RoboDK station: UR5Trajectory1.rdk

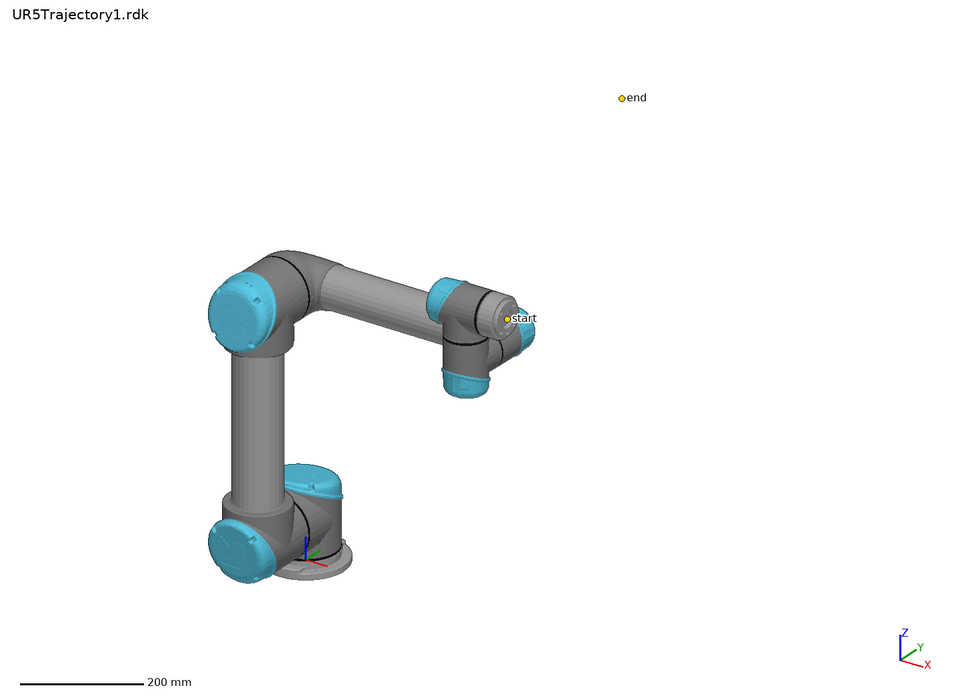
[picture v0: the station drawn from its stored meshes, robots at their saved joint values, targets as dots, program paths as lines]
Station 3TrajectoryUR5 (saved by RoboDK 5.6.8). Poses are relative to the parent item; angles as X-Y-Z fixed-axis rotations.
  - frame UR5 Base at (0, 0, 0) mm
    - robot UR5: 6 axes
        modified DH rows (alpha deg, a mm, theta deg, d mm): 0, 0, 0, 89.2; 90, 0, 180, 0; 0, 425, 0, 0; 0, 392, 0, 109.3; -90, 0, 0, 94.75; 90, 0, 180, 82.5
        joint limits [-360, -360, -360, -360, -360, -360] to [360, 360, 360, 360, 360, 360]; home [0, -90, -90, 0, 90, 0]; saved at [0, -90, -90, 0, 90, 0]
    - target end (Cartesian target) at (190.55, 618.42, 635.46) mm, rotated rx -81.71 ry 39.27 rz -77.04 deg; joints [90, -150, 10, 0, 10, 0] of UR5
    - target start (Cartesian target) at (474.5, -109.3, 608.95) mm, rotated rx -90 ry 0 rz -90 deg; joints [0, -90, -90, 0, 90, 0] of UR5
    - target Target1 (Cartesian target) at (190.55, 618.42, 635.46) mm, rotated rx -81.71 ry 39.27 rz -77.04 deg; joints [90, -150, 10, 0, 10, 0] of UR5
    - target Target2 (Cartesian target) at (190.55, 618.42, 635.46) mm, rotated rx -81.71 ry 39.27 rz -77.04 deg; joints [90, -140.405, -10, 10.405, 10, 0] of UR5
    - target Target3 (Cartesian target) at (190.55, 618.42, 635.46) mm, rotated rx -81.71 ry 39.27 rz -77.04 deg; joints [249.599, -53.819, 38.76, -178.356, -151.243, 27.758] of UR5
    - target Target4 (Cartesian target) at (190.55, 618.42, 635.46) mm, rotated rx -81.71 ry 39.27 rz -77.04 deg; joints [249.599, -16.687, -38.76, -137.968, -151.243, 27.758] of UR5
  - program Start->end1 (1 instructions, listed below)
  - program Start->end2 (1 instructions, listed below)
  - program Start->end3 (1 instructions, listed below)
  - program Start->end4 (1 instructions, listed below)
  - program moveL_Start->end (1 instructions, listed below)
  - program setup (2 instructions, listed below)

--- program Start->end1 (robot UR5) ---
  MoveJ (Target1)

--- program Start->end2 (robot UR5) ---
  MoveJ (Target2)

--- program Start->end3 (robot UR5) ---
  MoveJ (Target3)

--- program Start->end4 (robot UR5) ---
  MoveJ (Target4)

--- program moveL_Start->end (robot UR5) ---
  MoveL (Target4)

--- program setup (robot UR5) ---
  MoveJ (start)
  Set speed (10.0 mm/s)
